{attribute 'linkalways'} 
{attribute 'no_explicit_call' := 'This FB is a CLASS and must be accessed using methods or properties'}
{attribute 'enable_dynamic_creation'}
FUNCTION_BLOCK Node_F_VN_FindTemplateWalsh_AngleRange EXTENDS VisionNode
VAR
    ipSrcImage : _ITcVnImage;
    ipTemplateImage : _ITcVnImage;
	ipMatches : _ITcVnContainer;
	fMatchThreshold : _REAL(0.1);
	nProjections : _UDINT(10);
	fStartAngle : _LREAL(0);
	fStopAngle : _LREAL(1);
	nAngles : _UDINT(1);
    hrPrev : _HRESULT(S_OK);
	hresult : _HRESULT(S_OK);
END_VAR

METHOD PUBLIC  Clone : I_Node
VAR
	pNode : POINTER TO Node_F_VN_FindTemplateWalsh_AngleRange;
END_VAR
pNode := __NEW(Node_F_VN_FindTemplateWalsh_AngleRange);
Clone := pNode^;
END_METHOD

METHOD FB_init : BOOL
VAR_INPUT
	bInitRetains : BOOL; // if TRUE, the retain variables are initialized (warm start / cold start)
	bInCopyCode : BOOL;  // if TRUE, the instance afterwards gets moved into the copy code (online change)
END_VAR
AddInput('ipSrcImage', ipSrcImage);
AddInput('ipTemplateImage', ipTemplateImage);
AddInput('fMatchThreshold', fMatchThreshold);
AddInput('nProjections', nProjections);
AddInput('fStartAngle', fStartAngle);
AddInput('fStopAngle', fStopAngle);
AddInput('nAngles', nAngles);
AddInput('hrPrev', hrPrev);
AddOutput('ipMatches', ipMatches);
AddOutput('hresult',hresult);
END_METHOD

METHOD PROTECTED OnExecute
hresult.Value := F_VN_FindTemplateWalsh_AngleRange(
    ipSrcImage := ipSrcImage.Value,
    ipTemplateImage := ipTemplateImage.Value,
	ipMatches := ipMatches.Value,
	fMatchThreshold := fMatchThreshold.Value,
	nProjections := nProjections.Value,
	fStartAngle := fStartAngle.Value,
	fStopAngle := fStopAngle.Value,
	nAngles := nAngles.Value,
	hrPrev:= hrPrev.Value);
END_METHOD

METHOD PUBLIC PreExecutionCheck
VAR_INPUT
	Check : I_PreExecutionChecks;
END_VAR
Check.IsTrue(ipSrcImage.IsValid, 'ipSrcImage must contain an image');
Check.IsTrue(ipSrcImage.IsPixelDepth(8), 'ipSrcImage must be 8 or 32 bit pixel depth');
Check.IsTrue((ipSrcImage.HasChannelCount(1) OR ipSrcImage.HasChannelCount(3)), 'ipSrcImage must contain 1 or 3 channels');

Check.IsTrue((fMatchThreshold.Value >= 0 AND fMatchThreshold.Value <= 1), 'Threshold must be between 0..1, 1.0 would be a perfect match');
Check.IsTrue(nProjections.Value <= 50, 'The soft limit of 50 has been reached');

Check.IsTrue(ipTemplateImage.IsValid, 'ipTemplateImage must contain an image');
Check.IsTrue(ImagesHaveMatchingPixelFormats(ipSrcImage.Value, ipTemplateImage.Value), 'ipTemplateImage must have same pixel depth as ipSrcImage');
Check.IsTrue(ImagesHaveMatchingChannels(ipSrcImage.Value, ipTemplateImage.Value), 'ipTemplateImage must have same amount of channels as ipSrcImage');
Check.IsTrue(IsTemplateImageSmallerThanSourceImage(ipSrcImage.Value, ipTemplateImage.Value), 'ipTemplateImage must be smaller than ipSrcImage');
END_METHOD

END_FUNCTION_BLOCK

(* stored: Version 1.1.0.1, ProductVersion 3.1.4026.13
   POU Node_F_VN_FindTemplateWalsh_AngleRange: Id {0d677bf4-c205-0ed1-146c-9f1879b97175}, SpecialFunc None
   Folder Constructor: Id {a34c378b-cafc-0e80-0fa0-871365f4cd0a}
   Method Clone: Id {e133424c-84f8-04de-080f-86ad0c3de1fb}
   Method FB_init: Id {e51d7a39-bc2d-0e68-25c8-65633dda2edb}
   Method OnExecute: Id {cf77e752-749c-0624-2c01-34520b326d94}
   Method PreExecutionCheck: Id {c4b877a4-7ddd-0b3b-3d55-0aaeaf68af58} *)
